// Mitsubishi GX Developer project: パレット移載装置   PLC: Q02

PROGRAM INISAL
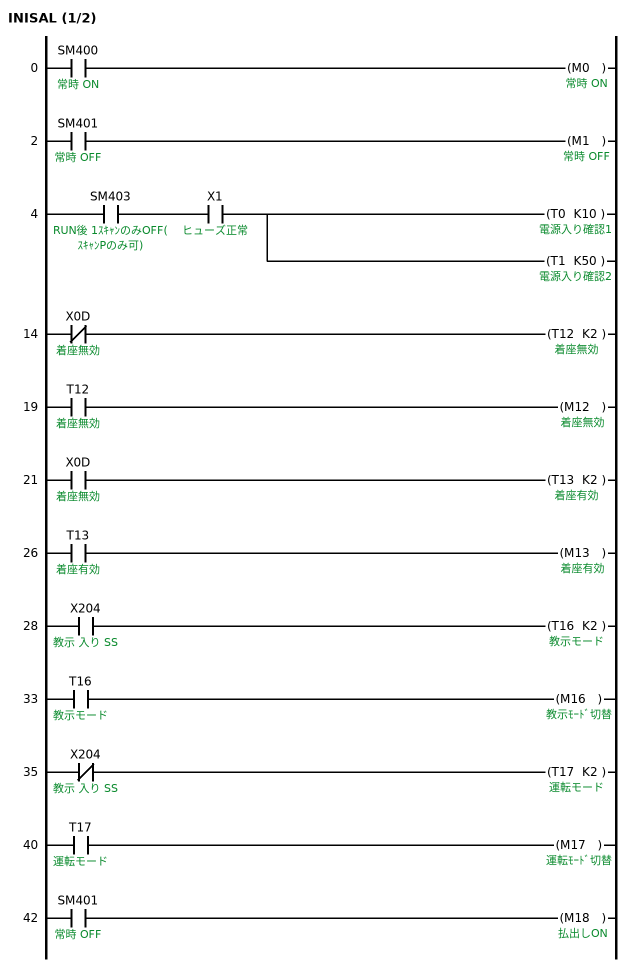
0     LD      SM400  ; 常時 ON
      OUT     M0  ; 常時 ON
2     LD      SM401  ; 常時 OFF
      OUT     M1  ; 常時 OFF
4     LD      SM403  ; RUN後 1ｽｷｬﾝのみOFF(ｽｷｬﾝPのみ可)
      AND     X1  ; ヒューズ正常
      OUT     T0 K10  ; 電源入り確認1
      OUT     T1 K50  ; 電源入り確認2
14    LDI     X0D  ; 着座無効
      OUT     T12 K2  ; 着座無効
19    LD      T12  ; 着座無効
      OUT     M12  ; 着座無効
21    LD      X0D  ; 着座無効
      OUT     T13 K2  ; 着座有効
26    LD      T13  ; 着座有効
      OUT     M13  ; 着座有効
28    LD      X204  ; 教示 入り SS
      OUT     T16 K2  ; 教示モード
33    LD      T16  ; 教示モード
      OUT     M16  ; 教示ﾓｰﾄﾞ切替
35    LDI     X204  ; 教示 入り SS
      OUT     T17 K2  ; 運転モード
40    LD      T17  ; 運転モード
      OUT     M17  ; 運転ﾓｰﾄﾞ切替
42    LD      SM401  ; 常時 OFF
      OUT     M18  ; 払出しON
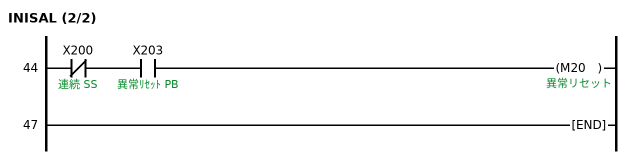
44    LDI     X200  ; 連続 SS
      AND     X203  ; 異常ﾘｾｯﾄ PB
      OUT     M20  ; 異常リセット
47    END
END_PROGRAM
